PROGRAM MAIN
VAR
	Flash: BLINK;
END_VAR

//Comms
Modbus_ReadInputs();
Modbus_WriteOutputs();
InputOutput();

//System
System();
Flash(ENABLE:= TRUE , TIMELOW:= T#500MS, TIMEHIGH:= T#500MS, OUT=> FlashBit);

END_PROGRAM

(* stored: Version 1.1.0.1, ProductVersion 3.1.4024.6
   POU MAIN: Id {7b8fc40a-e421-4ae3-8045-7a28ada69132}, SpecialFunc None *)
